{attribute addProperty BoxType "EP1122-0001-0017"}
{attribute addProperty Id "A_0026_EP1122_0001_0018A_0026_EP1122_0001_0018_D11347D11080068719478086"}
{attribute addProperty CRC "1817638569"}
{attribute addProperty SizeInBites "10800"}
{attribute addProperty SizeInBytes "68719478086"}
TYPE A_0025_EP1122_0001_0017_6C56F6A9 EXTENDS EP1122_179A0949 :
STRUCT
	{attribute addProperty Name "A_0026_EP1122_0001_0018"}
	A_0026_EP1122_0001_0018 : A_0026_EP1122_0001_0018_D11347D1;
END_STRUCT
END_TYPE

(* stored: Version 1.2.0.0, ProductVersion 3.1.4024.9
   DUT A_0025_EP1122_0001_0017_6C56F6A9: Id {5a2f04dd-36f5-409e-aaaa-c69911ae25d9} *)
